{attribute 'call_after_init'}
FUNCTION_BLOCK FB_MotionStageNC
VAR
    iMotionLogger : I_MotionLogger;
    {attribute 'no_copy'}
    AxisRef : REFERENCE TO AXIS_REF;
    {attribute 'no_copy'}
    stMotionEpicsItf : REFERENCE TO ST_MotionStage;
    iPersistentDataStorage : I_PersistentDataStorage;

    //Brakes : brake fb participate in sync comm with fbMotionDrive, fbMotionAxis and fbMotionInterlocks
    fbBrake : FB_BrakeNC := (BrakeMode := E_StageBrakeMode.IF_MOVING);
    // common interlocks
	{attribute 'pytmc' := 'pv:'}
    fbMotionInterlocksCommon : FB_MotionInterlocksCommon(iMotionLogger := iMotionLogger);
    // stage with Limit switches
    fbLimSwStatus : FB_LimSwStatus();
    fbMotionInterlocksLimSw : FB_MotionInterlocksLimSw ( iMotionInterlocksCommon:=fbMotionInterlocksCommon, iLimSwStatus:=fbLimSwStatus);
    fbHome : FB_HomeNC(AxisRef:=AxisRef, iMotionLogger:=iMotionLogger, iLimSwStatus:=fbLimSwStatus);;
    fbHalt : FB_HaltNC(AxisRef:=AxisRef);
    fbPower : FB_PowerNC(AxisRef:=AxisRef);
    fbReset : FB_ResetNC(AxisRef:=AxisRef);
    fbMoveAbsolute : FB_MoveAbsoluteNC(AxisRef:=AxisRef);
    fbAxisStatus : FB_AxisStatusNC(AxisRef:=AxisRef);
	{attribute 'pytmc' := 'pv:'}
    fbReadParameter : FB_ReadParameterNC(AxisRef:=AxisRef);
    fbWriteParameter  : FB_WriteParameterNC(AxisRef:=AxisRef);
    fbParamsSaveRestore: FB_ParamsSaveRestoreNC(AxisRef:=AxisRef, iPersistentDataStorage := iPersistentDataStorage);
	{attribute 'pytmc' := 'pv:'}
    fbEncoderScaling : FB_EncoderScaling();
	{attribute 'pytmc' := 'pv:'}
    fbBacklashCompensation : FB_BacklashCompensationNC(AxisRef:=AxisRef);
    fbMotionAxis : FB_MotionAxisNC(
        iHome := fbHome,
        iHalt := fbHalt,
        iPower := fbPower,
        iReset := fbReset,
        iMoveAbsolute := fbMoveAbsolute,
        iReadParameter := fbReadParameter,
        iWriteParameter  := fbWriteParameter,
        iParamSaveRestore:= fbParamsSaveRestore,
        iEncoderScaling := fbEncoderScaling,
        iAxisStatus := fbAxisStatus,
        iBacklashCompensation :=fbBacklashCompensation,
    );
    // Motion Requests
	{attribute 'pytmc' := 'pv:'}
    fbMoveRequest : FB_EpicsMoveRequest(stMotionEpicsItf:=stMotionEpicsItf);
    fbEpicsMotionParamsStatus : FB_EpicsMotionParamsStatus(stMotionEpicsItf:=stMotionEpicsItf);
    // Motion StateMachine
    fbStateMachine  : FB_MotionDriveStateMachine(
            iMotionAxis:=fbMotionAxis,
            iMoveRequest:=fbMoveRequest
    );

    fbMotionDrive: FB_MotionDrive (
        iBrake:=fbBrake,
        iMotionLogger:=iMotionLogger,
        iMotionInterlocks:=fbMotionInterlocksLimSw,
        iMotionAxis := fbMotionAxis,
        iMoveRequest := fbMoveRequest,
           iEpicsMotionParamsStatus := fbEpicsMotionParamsStatus,
        iMotionDriveStateMachine:=fbStateMachine
     ) ;
    // Drive Name
    {attribute 'hide'}
    sName : T_MaxString;
	bHomeCmd:BOOL;
	bMoveCmd:BOOL;
END_VAR

VAR_OUTPUT
    {attribute 'hide'}
	bMotionAxisError : BOOL;
    {attribute 'hide'}
	nMotionAxisErrorId : UDINT;
    {attribute 'hide'}
	bInterlocksError : BOOL;
    {attribute 'hide'}
	nInterlocksError : UDINT;
    {attribute 'hide'}
	eDriveState : E_MoveState;
    {attribute 'hide'}
	bDriveWatchDogStatus : BOOL;
    {attribute 'hide'}
	bAbortDone : BOOL;
    {attribute 'hide'}
	bAborted : BOOL;
    {attribute 'hide'}
	bLimHomeDone : BOOL;
END_VAR

IF NOT __ISVALIDREF(AxisRef) OR NOT __ISVALIDREF(stMotionEpicsItf)  THEN
	// Throw an exception here
    RETURN;
END_IF

IF bHomeCmd THEN
	THIS^.fbMoveRequest.HomeCmd := TRUE;
	bHomeCmd := FALSE;
ELSIF bMoveCmd THEN
	THIS^.fbMoveRequest.MoveCmd := TRUE;
	bMoveCmd:=FALSE;
END_IF

AxisRef.ReadStatus();

fbReset();
fbHalt();
fbPower();
fbBacklashCompensation();
fbMoveAbsolute();
fbHome();
fbAxisStatus();
fbReadParameter();
fbWriteParameter();
fbParamsSaveRestore();
fbMotionAxis();

fbLimSwStatus();
fbMotionInterlocksCommon();
fbMotionInterlocksLimSw();
fbMotionDrive();
fbMoveRequest();
fbStateMachine();
fbBrake();
fbEncoderScaling();
fbEpicsMotionParamsStatus();


bMotionAxisError := fbMotionAxis.Status.bError;
nMotionAxisErrorId := fbMotionAxis.Status.nErrorID;
bInterlocksError := fbMotionInterlocksCommon.Error;
nInterlocksError := fbMotionInterlocksCommon.ErrorID;
eDriveState := fbStateMachine.MoveState;
bAbortDone  := fbMotionAxis.Status.bAbortDone;
bAborted :=  fbAxisStatus.Aborted;
bLimHomeDone := fbMotionAxis.Status.bLimHomeDone;
bDriveWatchDogStatus := fbStateMachine.WatchDogStatus;

PROPERTY BrakeMode : E_StageBrakeMode
SET
fbBrake.BrakeMode := BrakeMode;
END_SET
END_PROPERTY

{attribute 'call_after_init'}
METHOD PRIVATE CallAfterInit
fbMotionInterlocksCommon.CallAfterInit(iMotionLogger := THIS^.iMotionLogger);
//fbLimSwStatus.CallAfterInit(iMotionLogger := THIS^.iMotionLogger);
fbMotionInterlocksLimSw.CallAfterInit(
        iMotionInterlocksCommon := THIS^.fbMotionInterlocksCommon,
        iLimSwStatus := THIS^.fbLimSwStatus
);

fbHome.CallAfterInit(
        AxisRef := THIS^.AxisRef,
        iMotionLogger := THIS^.iMotionLogger,
        iLimSwStatus := THIS^.fbLimSwStatus
);

fbHalt.CallAfterInit(AxisRef := THIS^.AxisRef);
fbPower.CallAfterInit(AxisRef := THIS^.AxisRef);
fbReset.CallAfterInit(AxisRef := THIS^.AxisRef);
fbMoveAbsolute.CallAfterInit(AxisRef := THIS^.AxisRef);
fbReadParameter.CallAfterInit(AxisRef:=THIS^.AxisRef);
fbWriteParameter.CallAfterInit(AxisRef:=THIS^.AxisRef);

fbParamsSaveRestore.CallAfterInit(
        AxisRef := THIS^.AxisRef,
        iPersistentDataStorage := THIS^.iPersistentDataStorage
);

// Pass correctly initialized Motion axis status dependencies
fbAxisStatus.CallAfterInit(AxisRef := THIS^.AxisRef);
fbBacklashCompensation.CallAfterInit(AxisRef := THIS^.AxisRef);

// Pass correctly initialized Motion axis dependencies
fbMotionAxis.CallAfterInit(
        iHome := THIS^.fbHome,
        iHalt := THIS^.fbHalt,
        iPower := THIS^.fbPower,
        iReset := THIS^.fbReset,
        iMoveAbsolute := THIS^.fbMoveAbsolute,
        iReadParameter := THIS^.fbReadParameter,
        iWriteParameter  := THIS^.fbWriteParameter,
        iParamSaveRestore:= THIS^.fbParamsSaveRestore,
        iEncoderScaling := THIS^.fbEncoderScaling,
        iAxisStatus := THIS^.fbAxisStatus,
        iBacklashCompensation := THIS^.fbBacklashCompensation
);

fbMoveRequest.CallAfterInit(stMotionEpicsItf:= THIS^.stMotionEpicsItf);
fbEpicsMotionParamsStatus.CallAfterInit(stMotionEpicsItf:= THIS^.stMotionEpicsItf);
fbStateMachine.CallAfterInit(iMotionAxis:=fbMotionAxis, iMoveRequest:=fbMoveRequest);
// Pass correctly initialized drive dependencies
fbMotionDrive.CallAfterInit(
     iBrake:=THIS^.fbBrake,
     iMotionInterlocks:=THIS^.fbMotionInterlocksLimSw,
     iMotionLogger:=THIS^.iMotionLogger,
     iMotionAxis:=THIS^.fbMotionAxis,
     iMoveRequest:=THIS^.fbMoveRequest,
     iEpicsMotionParamsStatus:=THIS^.fbEpicsMotionParamsStatus,
     iMotionDriveStateMachine:=THIS^.fbStateMachine
);

THIS^.stMotionEpicsItf.sName := THIS^.sName;
END_METHOD

METHOD INTERNAL EnableBacklashCompensation
VAR_INPUT
    UserEnable : BOOL;
    Compensation : LREAL;
END_VAR
THIS^.fbBacklashCompensation.EnableBacklashCompensation(UserEnable:=UserEnable, Compensation:=Compensation);
END_METHOD

PROPERTY EnableMode : E_StageEnableMode
SET
fbMoveRequest.EnableMode := EnableMode;
END_SET
END_PROPERTY

//FB_Init is always available implicitly and it is used primarily for initialization.
//The return value is not evaluated. For a specific influence, you can also declare the
//methods explicitly and provide additional code there with the standard initialization
//code. You can evaluate the return value.
METHOD FB_Init: BOOL
VAR_INPUT
    bInitRetains: BOOL; // TRUE: the retain variables are initialized (reset warm / reset cold)
    bInCopyCode: BOOL;  // TRUE: the instance will be copied to the copy code afterward (online change)
    iMotionLogger : I_MotionLogger;
    AxisRef : REFERENCE TO AXIS_REF;
    stMotionEpicsItf : REFERENCE TO ST_MotionStage;
    iPersistentDataStorage : I_PersistentDataStorage;
    sName : T_MaxString;
END_VAR
THIS^.iMotionLogger := iMotionLogger;
THIS^.AxisRef REF= AxisRef;
THIS^.iPersistentDataStorage := iPersistentDataStorage;
THIS^.stMotionEpicsItf REF=stMotionEpicsItf;
THIS^.sName := sName;
END_METHOD

PROPERTY HardwareEnable : BOOL
SET
fbMotionInterlocksCommon.HardwareEnable := HardwareEnable;
END_SET
END_PROPERTY

PROPERTY HomeMode : E_EpicsHomeCmd
SET
fbHome.Mode := HomeMode;
fbMoveRequest.HomeMode := HomeMode;
END_SET
END_PROPERTY

PROPERTY LimBackward : BOOL
SET
THIS^.fbLimSwStatus.LimBackward := LimBackward;
END_SET
END_PROPERTY

PROPERTY LimForward : BOOL
SET
THIS^.fbLimSwStatus.LimForward := LimForward;
END_SET
END_PROPERTY

PROPERTY LimHome : BOOL
SET
THIS^.fbLimSwStatus.LimHome:= LimHome;
END_SET
END_PROPERTY

METHOD INTERNAL UserCmds
VAR_INPUT
	MoveCmd : BOOL;
	HomeCmd : BOOL;
END_VAR
THIS^.fbMoveRequest.MoveCmd := MoveCmd;
THIS^.fbMoveRequest.HomeCmd := HomeCmd;
END_METHOD

PROPERTY UserEnable : BOOL
SET
THIS^.fbMotionInterlocksCommon.UserEnable := UserEnable;
END_SET
END_PROPERTY

END_FUNCTION_BLOCK

(* stored: Version 1.1.0.1
   POU FB_MotionStageNC: Id {27a9489d-ed3b-4885-89cd-bbc7b70f9440}, SpecialFunc None
   Property BrakeMode: Id {7b563b76-fecc-4885-824b-f91a0bc21af3}
   Set Set: Id {15a41f16-798f-4b50-9250-e347873647b8}
   Method CallAfterInit: Id {e7a5e1c3-8324-4257-a302-ab714cb009e4}
   Method EnableBacklashCompensation: Id {87740abd-9537-43e7-9863-d2436efc09c8}
   Property EnableMode: Id {d2517567-d217-491d-9b68-9264f829d81e}
   Set Set: Id {1782045b-083a-4984-8c31-ce01cd3f2942}
   Method FB_Init: Id {fe4c9de1-abf0-4550-ae13-2cd56df378be}
   Property HardwareEnable: Id {de413790-64d6-4df7-be45-e16e9a7af71c}
   Set Set: Id {4e90c6a1-868e-40b9-a14d-f0f664cb75ae}
   Property HomeMode: Id {6fbba694-14cc-47d7-b386-b3a87f93d4ab}
   Set Set: Id {1a6336ac-7eec-4dce-ac7d-8543b797a82e}
   Property LimBackward: Id {0a694a2c-821b-487b-b05f-33f0c7db41ce}
   Set Set: Id {da6b1409-3d4c-4a22-9e2d-f94bf698dc21}
   Property LimForward: Id {12e7d2e2-4178-42bf-a874-e4fbc8f61cdb}
   Set Set: Id {3d00e8a0-812a-46a2-abcc-4f40ba55e42d}
   Property LimHome: Id {f54a4acf-f180-407e-8cce-8faeca002258}
   Set Set: Id {e51dc72a-5425-479a-b339-56588f629df8}
   Method UserCmds: Id {11a63b1a-6a72-4e18-b829-4ce12aeabb4f}
   Property UserEnable: Id {863b6547-890c-46aa-afec-34d889e5d2ed}
   Set Set: Id {a26c7d34-2d19-4d31-8732-6c1180f87277} *)
